	IO6 : NOP   0;
	      NOP   0;
	// --- FCM 07 - Recycling air flap ---
	    L "MAL1S032Par".Ilo.ILOMode;
	    L  7;
	    <>I;
	    SPB IO7;
	// man on
	      U     "MAL1S032Par".Ilo.GrCMDManOn[1];
	      S     "G273M".Gr.InManual; // RECYCLING AIR LOUVER KILN 1
	      S     "G278M".Gr.InManual; // WITHERING AIR KILN 1
	      R     "MAL1S032Par".Ilo.GrCMDManOn[1];
	// man off
	      U     "MAL1S032Par".Ilo.GrCMDManOff[1];
	      S     "G273M".Gr.CmdManualOff; // RECYCLING AIR LOUVER KILN 1
	      R     "G273M".Gr.InManual; // RECYCLING AIR LOUVER KILN 1
	      R     "G273M".USW14; // ILO-cmd
	      R     "G273M".USW15; // ILO-cmd
	      S     "G278M".Gr.CmdManualOff; // WITHERING AIR KILN 1
	      R     "G278M".Gr.InManual; // WITHERING AIR KILN 1
	      R     "G278M".USW14; // ILO-cmd
	      R     "G278M".USW15; // ILO-cmd
	      R     "MAL1S032Par".Ilo.GrCMDManOff[1];
	      R     "MAL1S032Par".Ilo.GrCMDManAdditional.Cmd1[1];
	      R     "MAL1S032Par".Ilo.GrCMDManAdditional.Cmd2[1];
	// man start
	      U     "MAL1S032Par".Ilo.GrCMDManStart[1];
	      S     "G273M".Gr.CmdOn; // RECYCLING AIR LOUVER KILN 1
	      S     "G273M".Gr.CmdContinue; // RECYCLING AIR LOUVER KILN 1
	      S     "G278M".Gr.CmdOn; // WITHERING AIR KILN 1
	      S     "G278M".Gr.CmdContinue; // WITHERING AIR KILN 1
	      R     "MAL1S032Par".Ilo.GrCMDManStart[1];
	      U     "MAL1S032Par".Ilo.GrCMDManStart[2];
	      R     "MAL1S032Par".Ilo.GrCMDManStart[2];
	// man stop
	      U     "MAL1S032Par".Ilo.GrCMDManStop[1];
	      S     "G273M".Gr.CmdOff; // RECYCLING AIR LOUVER KILN 1
	      S     "G278M".Gr.CmdOff; // WITHERING AIR KILN 1
	      R     "MAL1S032Par".Ilo.GrCMDManStop[1];
	// man fault reset
	      U     "MAL1S032Par".Ilo.GrCMDManFaultReset[1];
	      S     "G273M".Gr.CmdFaultReset; // RECYCLING AIR LOUVER KILN 1
	      S     "G278M".Gr.CmdFaultReset; // WITHERING AIR KILN 1
	      R     "MAL1S032Par".Ilo.GrCMDManFaultReset[1];
	// moving direction
	//
	// target position
	      UN    "G273M".Gr.InManual; // RECYCLING AIR LOUVER KILN 1
	      SPB   F07a;
	      L     "MAL1S032Par".Ilo.SetpointInt01[1];
	      T     "MAL1S032Par".Par.ParIntProcess.TarPos_ILO_RecycAir;
	F07a:  NOP   0;
	IO7 : NOP   0;
	      NOP   0;
	// --- FCM 09 - Floor drives ---
	    L "MAL1S032Par".Ilo.ILOMode;
	    L  9;
	    <>I;
	    SPB IO9;
	// man on
	      U     "MAL1S032Par".Ilo.GrCMDManOn[1];
	      S     "G266M".Gr.InManual; // TRAVELLING DRIVE KILN 1
	      R     "MAL1S032Par".Ilo.GrCMDManOn[1];
	// man off
	      U     "MAL1S032Par".Ilo.GrCMDManOff[1];
	      S     "G266M".Gr.CmdManualOff; // TRAVELLING DRIVE KILN 1
	      R     "G266M".Gr.InManual; // TRAVELLING DRIVE KILN 1
	      R     "G266M".USW14; // ILO-cmd
	      R     "G266M".USW15; // ILO-cmd
	      R     "MAL1S032Par".Ilo.GrCMDManOff[1];
	      R     "MAL1S032Par".Ilo.GrCMDManAdditional.Cmd1[1];
	      R     "MAL1S032Par".Ilo.GrCMDManAdditional.Cmd2[1];
	// man start
	      U     "MAL1S032Par".Ilo.GrCMDManStart[1];
	      S     "G266M".Gr.CmdOn; // TRAVELLING DRIVE KILN 1
	      S     "G266M".Gr.CmdContinue; // TRAVELLING DRIVE KILN 1
	      R     "MAL1S032Par".Ilo.GrCMDManStart[1];
	      U     "MAL1S032Par".Ilo.GrCMDManStart[2];
	      R     "MAL1S032Par".Ilo.GrCMDManStart[2];
	// man stop
	      U     "MAL1S032Par".Ilo.GrCMDManStop[1];
	      S     "G266M".Gr.CmdOff; // TRAVELLING DRIVE KILN 1
	      R     "MAL1S032Par".Ilo.GrCMDManStop[1];
	// man fault reset
	      U     "MAL1S032Par".Ilo.GrCMDManFaultReset[1];
	      S     "G266M".Gr.CmdFaultReset; // TRAVELLING DRIVE KILN 1
	      R     "MAL1S032Par".Ilo.GrCMDManFaultReset[1];
	f091: NOP   0;
	      UN    "G266M".Gr.InManual; // TRAVELLING DRIVE KILN 1
	      O     ;
	      UN    "MAL1S032Par".Ilo.GrCMDManAdditional.Cmd1[1];
	      UN    "MAL1S032Par".Ilo.GrCMDManAdditional.Cmd2[1];
	      SPB   f092;
	      U     "MAL1S032Par".Ilo.GrCMDManAdditional.Cmd1[1];
	      =     "G266M".USW14; // ILO-cmd run fwd
	      U     "MAL1S032Par".Ilo.GrCMDManAdditional.Cmd2[1];
	      =     "G266M".USW15; // ILO-cmd run rev
	// target position
	      L     "MAL1S032Par".Ilo.SetpointInt01[1];
	      T     "MAL1S032Par".Par.ParIntProcess.Speed_ILO_FloorRotating;
	f092: NOP   0;

	IO9 : NOP   0;
	      NOP   0;
	// --- FCM 10 - Floor drives and lifting devices ---
	    L "MAL1S032Par".Ilo.ILOMode;
	    L  10;
	    <>I;
	    SPB IO10;
	// man on
	      U     "MAL1S032Par".Ilo.GrCMDManOn[1];
	      S     "G265M".Gr.InManual; // LIFTING DEVICE KILN 1
	      S     "G265M".Gr.CmdOn; // No Button: LIFTING DEVICE KILN 1
	      S     "G265M".Gr.CmdContinue; // No Button LIFTING DEVICE KILN 1
	      S     "G266M".Gr.InManual; // TRAVELLING DRIVE KILN 1
	      R     "MAL1S032Par".Ilo.GrCMDManOn[1];
	// man off
	      U     "MAL1S032Par".Ilo.GrCMDManOff[1];
	      S     "G265M".Gr.CmdManualOff; // LIFTING DEVICE KILN 1
	      R     "G265M".Gr.InManual; // LIFTING DEVICE KILN 1
	      R     "G265M".USW14; // ILO-cmd
	      R     "G265M".USW15; // ILO-cmd
	      S     "G266M".Gr.CmdManualOff; // TRAVELLING DRIVE KILN 1
	      R     "G266M".Gr.InManual; // TRAVELLING DRIVE KILN 1
	      R     "G266M".USW14; // ILO-cmd
	      R     "G266M".USW15; // ILO-cmd
	      R     "MAL1S032Par".Ilo.GrCMDManOff[1];
	      R     "MAL1S032Par".Ilo.GrCMDManAdditional.Cmd1[1];
	      R     "MAL1S032Par".Ilo.GrCMDManAdditional.Cmd2[1];
	// man start
	      U     "MAL1S032Par".Ilo.GrCMDManStart[1];
	      S     "G266M".Gr.CmdOn; // TRAVELLING DRIVE KILN 1
	      S     "G266M".Gr.CmdContinue; // TRAVELLING DRIVE KILN 1
	      R     "MAL1S032Par".Ilo.GrCMDManStart[1];
	      U     "MAL1S032Par".Ilo.GrCMDManStart[2];
	      S     "G265M".Gr.CmdOn; // LIFTING DEVICE KILN 1
	      S     "G265M".Gr.CmdContinue; // LIFTING DEVICE KILN 1
	      R     "MAL1S032Par".Ilo.GrCMDManStart[2];
	      U     "MAL1S032Par".Ilo.GrCMDManStart[3];
	      R     "MAL1S032Par".Ilo.GrCMDManStart[3];
	// man stop
	      U     "MAL1S032Par".Ilo.GrCMDManStop[1];
	      S     "G265M".Gr.CmdOff; // LIFTING DEVICE KILN 1
	      S     "G266M".Gr.CmdOff; // TRAVELLING DRIVE KILN 1
	      R     "MAL1S032Par".Ilo.GrCMDManStop[1];
	// man fault reset
	      U     "MAL1S032Par".Ilo.GrCMDManFaultReset[1];
	      S     "G265M".Gr.CmdFaultReset; // LIFTING DEVICE KILN 1
	      S     "G266M".Gr.CmdFaultReset; // TRAVELLING DRIVE KILN 1
	      R     "MAL1S032Par".Ilo.GrCMDManFaultReset[1];
	// moving direction
	f101: NOP   0;
	      UN    "G266M".Gr.InManual; // TRAVELLING DRIVE KILN 1
	      O     ;
	      UN    "MAL1S032Par".Ilo.GrCMDManAdditional.Cmd1[1];
	      UN    "MAL1S032Par".Ilo.GrCMDManAdditional.Cmd2[1];
	      SPB   f102;
	      U     "MAL1S032Par".Ilo.GrCMDManAdditional.Cmd1[1];
	      =     "G266M".USW14; // ILO-cmd run fwd
	      U     "MAL1S032Par".Ilo.GrCMDManAdditional.Cmd2[1];
	      =     "G266M".USW15; // ILO-cmd run rev
	// target speed floor drives
	      L     "MAL1S032Par".Ilo.SetpointInt01[1];
	      T     "MAL1S032Par".Par.ParIntProcess.Speed_ILO_FloorRotating;
	f102: NOP   0;
	      UN    "G265M".Gr.InManual; // LIFTING DEVICE KILN 1
	      O(    ;
	      L     "MAL1S032Par".Ilo.Code_ILO_Funktion0;
	      L     1000;
	      <>I   ;
	      )     ;
	      SPB   f103;
	// target position lifting devices
	      L     "MAL1S032Par".Ilo.SetpointInt02[1];
	      T     "MAL1S032Par".Par.ParIntProcess.TarPos_ILO_LiftDev;
	f103: NOP   0;

	IO10 : NOP   0;
	      NOP   0;
	// --- FCM 11 - Floor drives and lifting devices and screw ---
	    L "MAL1S032Par".Ilo.ILOMode;
	    L  11;
	    <>I;
	    SPB IO11;
	// man on
	      U     "MAL1S032Par".Ilo.GrCMDManOn[1];
	      S     "G265M".Gr.InManual; // LIFTING DEVICE KILN 1
	      S     "G265M".Gr.CmdOn; // No Button: LIFTING DEVICE KILN 1
	      S     "G265M".Gr.CmdContinue; // No Button LIFTING DEVICE KILN 1
	      S     "G266M".Gr.InManual; // TRAVELLING DRIVE KILN 1
	      S     "G267M".Gr.InManual; // UNLOADING / LOADING SCREW KILN 1
	      R     "MAL1S032Par".Ilo.GrCMDManOn[1];
	// man off
	      U     "MAL1S032Par".Ilo.GrCMDManOff[1];
	      S     "G265M".Gr.CmdManualOff; // LIFTING DEVICE KILN 1
	      R     "G265M".Gr.InManual; // LIFTING DEVICE KILN 1
	      R     "G265M".USW14; // ILO-cmd
	      R     "G265M".USW15; // ILO-cmd
	      S     "G266M".Gr.CmdManualOff; // TRAVELLING DRIVE KILN 1
	      R     "G266M".Gr.InManual; // TRAVELLING DRIVE KILN 1
	      R     "G266M".USW14; // ILO-cmd
	      R     "G266M".USW15; // ILO-cmd
	      S     "G267M".Gr.CmdManualOff; // UNLOADING / LOADING SCREW KILN 1
	      R     "G267M".Gr.InManual; // UNLOADING / LOADING SCREW KILN 1
	      R     "G267M".USW14; // ILO-cmd
	      R     "G267M".USW15; // ILO-cmd
	      R     "MAL1S032Par".Ilo.GrCMDManOff[1];
	      R     "MAL1S032Par".Ilo.GrCMDManAdditional.Cmd1[1];
	      R     "MAL1S032Par".Ilo.GrCMDManAdditional.Cmd2[1];
	// man start
	      U     "MAL1S032Par".Ilo.GrCMDManStart[1];
	      S     "G266M".Gr.CmdOn; // TRAVELLING DRIVE KILN 1
	      S     "G266M".Gr.CmdContinue; // TRAVELLING DRIVE KILN 1
	      R     "MAL1S032Par".Ilo.GrCMDManStart[1];
	      U     "MAL1S032Par".Ilo.GrCMDManStart[2];
	      S     "G265M".Gr.CmdOn; // LIFTING DEVICE KILN 1
	      S     "G265M".Gr.CmdContinue; // LIFTING DEVICE KILN 1
	      R     "MAL1S032Par".Ilo.GrCMDManStart[2];
	      U     "MAL1S032Par".Ilo.GrCMDManStart[3];
	      S     "G267M".Gr.CmdOn; // UNLOADING / LOADING SCREW KILN 1
	      S     "G267M".Gr.CmdContinue; // UNLOADING / LOADING SCREW KILN 1
	      R     "MAL1S032Par".Ilo.GrCMDManStart[3];
	      U     "MAL1S032Par".Ilo.GrCMDManStart[4];
	      S     "G267M".Gr.CmdOn; // UNLOADING / LOADING SCREW KILN 1
	      S     "G267M".Gr.CmdContinue; // UNLOADING / LOADING SCREW KILN 1
	      R     "MAL1S032Par".Ilo.GrCMDManStart[4];
	// man stop
	      U     "MAL1S032Par".Ilo.GrCMDManStop[1];
	      S     "G265M".Gr.CmdOff; // LIFTING DEVICE KILN 1
	      S     "G266M".Gr.CmdOff; // TRAVELLING DRIVE KILN 1
	      S     "G267M".Gr.CmdOff; // UNLOADING / LOADING SCREW KILN 1
	      R     "MAL1S032Par".Ilo.GrCMDManStop[1];
	// man fault reset
	      U     "MAL1S032Par".Ilo.GrCMDManFaultReset[1];
	      S     "G265M".Gr.CmdFaultReset; // LIFTING DEVICE KILN 1
	      S     "G266M".Gr.CmdFaultReset; // TRAVELLING DRIVE KILN 1
	      S     "G267M".Gr.CmdFaultReset; // UNLOADING / LOADING SCREW KILN 1
	      R     "MAL1S032Par".Ilo.GrCMDManFaultReset[1];
	// moving direction
	      UN    "G266M".Gr.InManual; // TRAVELLING DRIVE KILN 1
	      O     ;
	      UN    "MAL1S032Par".Ilo.GrCMDManAdditional.Cmd1[1];
	      UN    "MAL1S032Par".Ilo.GrCMDManAdditional.Cmd2[1];
	      SPB   f112;
	      U     "MAL1S032Par".Ilo.GrCMDManAdditional.Cmd1[1];
	      =     "G266M".USW14; // ILO-cmd run fwd
	      U     "MAL1S032Par".Ilo.GrCMDManAdditional.Cmd2[1];
	      =     "G266M".USW15; // ILO-cmd run rev
	// target speed floor drives
	      L     "MAL1S032Par".Ilo.SetpointInt01[1];
	      T     "MAL1S032Par".Par.ParIntProcess.Speed_ILO_FloorRotating;
	f112: NOP   0;
	      UN    "G265M".Gr.InManual; // Malting Plant OAO Belsolod Ivanonvo Weissrussland
	      O(    ;
	      L     "MAL1S032Par".Ilo.Code_ILO_Funktion0;
	      L     1100;
	      <>I   ;
	      )     ;
	      SPB   f113;
	// target position lifting devices
	      L     "MAL1S032Par".Ilo.SetpointInt01[2];
	      L     "MAL1S032Par".Ilo.SetpointInt02[1];
	      T     "MAL1S032Par".Par.ParIntProcess.TarPos_ILO_LiftDev;
	f113: NOP   0;
	      UN    "G267M".Gr.InManual; // UNLOADING / LOADING SCREW KILN 1
	      O     ;
	      UN    "MAL1S032Par".Ilo.GrCMDManAdditional.Cmd1[3];
	      UN    "MAL1S032Par".Ilo.GrCMDManAdditional.Cmd2[3];
	      SPB   f114;
	      U     "MAL1S032Par".Ilo.GrCMDManAdditional.Cmd1[3];
	      =     "G267M".USW14; // ILO-cmd run fwd
	      U     "MAL1S032Par".Ilo.GrCMDManAdditional.Cmd2[3];
	      =     "G267M".USW15; // ILO-cmd run rev
	f114: NOP   0;
	IO11 : NOP   0;
	      NOP   0;
	// --- FCM 12 - Floor drives and lifting devices and screw and discharging flap ---
	    L "MAL1S032Par".Ilo.ILOMode;
	    L  12;
	    <>I;
	    SPB IO12;
	// man on
	      U     "MAL1S032Par".Ilo.GrCMDManOn[1];
	      S     "G265M".Gr.InManual; // LIFTING DEVICE KILN 1
	      S     "G265M".Gr.CmdOn; // No Button: LIFTING DEVICE KILN 1
	      S     "G265M".Gr.CmdContinue; // No Button LIFTING DEVICE KILN 1
	      S     "G266M".Gr.InManual; // TRAVELLING DRIVE KILN 1
	      S     "G267M".Gr.InManual; // UNLOADING / LOADING SCREW KILN 1
	      S     "G268M".Gr.InManual; // DISCHARGE DOOR KILN 1
	      R     "MAL1S032Par".Ilo.GrCMDManOn[1];
	// man off
	      U     "MAL1S032Par".Ilo.GrCMDManOff[1];
	      S     "G265M".Gr.CmdManualOff; // LIFTING DEVICE KILN 1
	      R     "G265M".Gr.InManual; // LIFTING DEVICE KILN 1
	      R     "G265M".USW14; // ILO-cmd
	      R     "G265M".USW15; // ILO-cmd
	      S     "G266M".Gr.CmdManualOff; // TRAVELLING DRIVE KILN 1
	      R     "G266M".Gr.InManual; // TRAVELLING DRIVE KILN 1
	      R     "G266M".USW14; // ILO-cmd
	      R     "G266M".USW15; // ILO-cmd
	      S     "G267M".Gr.CmdManualOff; // UNLOADING / LOADING SCREW KILN 1
	      R     "G267M".Gr.InManual; // UNLOADING / LOADING SCREW KILN 1
	      R     "G267M".USW14; // ILO-cmd
	      R     "G267M".USW15; // ILO-cmd
	      S     "G268M".Gr.CmdManualOff; // DISCHARGE DOOR KILN 1
	      R     "G268M".Gr.InManual; // DISCHARGE DOOR KILN 1
	      R     "G268M".USW14; // ILO-cmd
	      R     "G268M".USW15; // ILO-cmd
	      R     "MAL1S032Par".Ilo.GrCMDManOff[1];
	      R     "MAL1S032Par".Ilo.GrCMDManAdditional.Cmd1[1];
	      R     "MAL1S032Par".Ilo.GrCMDManAdditional.Cmd2[1];
	// man start
	      U     "MAL1S032Par".Ilo.GrCMDManStart[1];
	      S     "G266M".Gr.CmdOn; // TRAVELLING DRIVE KILN 1
	      S     "G266M".Gr.CmdContinue; // TRAVELLING DRIVE KILN 1
	      R     "MAL1S032Par".Ilo.GrCMDManStart[1];
	      U     "MAL1S032Par".Ilo.GrCMDManStart[2];
	      S     "G265M".Gr.CmdOn; // LIFTING DEVICE KILN 1
	      S     "G265M".Gr.CmdContinue; // LIFTING DEVICE KILN 1
	      R     "MAL1S032Par".Ilo.GrCMDManStart[2];
	      U     "MAL1S032Par".Ilo.GrCMDManStart[3];
	      S     "G267M".Gr.CmdOn; // UNLOADING / LOADING SCREW KILN 1
	      S     "G267M".Gr.CmdContinue; // UNLOADING / LOADING SCREW KILN 1
	      R     "MAL1S032Par".Ilo.GrCMDManStart[3];
	      U     "MAL1S032Par".Ilo.GrCMDManStart[4];
	      S     "G267M".Gr.CmdOn; // UNLOADING / LOADING SCREW KILN 1
	      S     "G267M".Gr.CmdContinue; // UNLOADING / LOADING SCREW KILN 1
	      R     "MAL1S032Par".Ilo.GrCMDManStart[4];
	// man stop
	      U     "MAL1S032Par".Ilo.GrCMDManStop[1];
	      S     "G265M".Gr.CmdOff; // LIFTING DEVICE KILN 1
	      S     "G266M".Gr.CmdOff; // TRAVELLING DRIVE KILN 1
	      S     "G267M".Gr.CmdOff; // UNLOADING / LOADING SCREW KILN 1
	      S     "G268M".Gr.CmdOff; // DISCHARGE DOOR KILN 1
	      R     "MAL1S032Par".Ilo.GrCMDManStop[1];
	// man fault reset
	      U     "MAL1S032Par".Ilo.GrCMDManFaultReset[1];
	      S     "G265M".Gr.CmdFaultReset; // LIFTING DEVICE KILN 1
	      S     "G266M".Gr.CmdFaultReset; // TRAVELLING DRIVE KILN 1
	      S     "G267M".Gr.CmdFaultReset; // UNLOADING / LOADING SCREW KILN 1
	      S     "G268M".Gr.CmdFaultReset; // DISCHARGE DOOR KILN 1
	      R     "MAL1S032Par".Ilo.GrCMDManFaultReset[1];
	// moving direction
	      UN    "G266M".Gr.InManual; // TRAVELLING DRIVE KILN 1
	      O     ;
	      UN    "MAL1S032Par".Ilo.GrCMDManAdditional.Cmd1[1];
	      UN    "MAL1S032Par".Ilo.GrCMDManAdditional.Cmd2[1];
	      SPB   f122;
	      U     "MAL1S032Par".Ilo.GrCMDManAdditional.Cmd1[1];
	      =     "G266M".USW14; // ILO-cmd run fwd
	      U     "MAL1S032Par".Ilo.GrCMDManAdditional.Cmd2[1];
	      =     "G266M".USW15; // ILO-cmd run rev
	// target speed floor drives
	      L     "MAL1S032Par".Ilo.SetpointInt01[1];
	      T     "MAL1S032Par".Par.ParIntProcess.Speed_ILO_FloorRotating;
	f122: NOP   0;
	      UN    "G265M".Gr.InManual; // LIFTING DEVICE KILN 1
	      O(    ;
	      L     "MAL1S032Par".Ilo.Code_ILO_Funktion0;
	      L     1200;
	      <>I   ;
	      )     ;
	      SPB   f123;
	// target position lifting devices
	      L     "MAL1S032Par".Ilo.SetpointInt02[1];
	      T     "MAL1S032Par".Par.ParIntProcess.TarPos_ILO_LiftDev;
	f123: NOP   0;
	      UN    "G267M".Gr.InManual; // Malting Plant OAO Belsolod Ivanonvo Weissrussland
	      O     ;
	      UN    "MAL1S032Par".Ilo.GrCMDManAdditional.Cmd1[3];
	      UN    "MAL1S032Par".Ilo.GrCMDManAdditional.Cmd2[3];
	      SPB   f124;
	      U     "MAL1S032Par".Ilo.GrCMDManAdditional.Cmd1[3];
	      =     "G267M".USW14; // ILO-cmd run fwd
	      U     "MAL1S032Par".Ilo.GrCMDManAdditional.Cmd2[3];
	      =     "G267M".USW15; // ILO-cmd run rev
	f124: NOP   0;
	      UN    "G268M".Gr.InManual; // DISCHARGE DOOR KILN 1
	      O     ;
	      UN    "MAL1S032Par".Ilo.GrCMDManAdditional.Cmd1[4];
	      UN    "MAL1S032Par".Ilo.GrCMDManAdditional.Cmd2[4];
	      SPB   f125;
	      U     "MAL1S032Par".Ilo.GrCMDManAdditional.Cmd1[4];
	      =     "G268M".USW14; // ILO-cmd OPEN
	      U     "MAL1S032Par".Ilo.GrCMDManAdditional.Cmd2[4];
	      =     "G268M".USW15; // ILO-cmd CLOSE
	f125: NOP   0;
	IO12 : NOP   0;
	//
	// copy state
	      U     "G265M".Gr.InOutAutostartMan; // LIFTING DEVICE KILN 1
	      =     "MAL1S032Par".Ilo.GrSTMan[1];
	      U     "G266M".Gr.InOutAutostartMan; // TRAVELLING DRIVE KILN 1
	      =     "MAL1S032Par".Ilo.GrSTMan[2];
	      U     "G267M".Gr.InOutAutostartMan; // UNLOADING / LOADING SCREW KILN 1
	      =     "MAL1S032Par".Ilo.GrSTMan[3];
	      U     "G268M".Gr.InOutAutostartMan; // DISCHARGE DOOR KILN 1
	      =     "MAL1S032Par".Ilo.GrSTMan[4];
	      U     "G271M".Gr.InOutAutostartMan; // FAN KILN 1
	      =     "MAL1S032Par".Ilo.GrSTMan[6];
	      U     "G276M".Gr.InOutAutostartMan; // HEATING KILN 1
	      =     "MAL1S032Par".Ilo.GrSTMan[11];
	      U     "G277M".Gr.InOutAutostartMan; // LOUVER AIR HEATER 1 FOR KILN 1
	      =     "MAL1S032Par".Ilo.GrSTMan[12];
	      U     "G272M".Gr.InOutAutostartMan; // FRESH AIR LOUVER KILN 1
	      =     "MAL1S032Par".Ilo.GrSTMan[13];
	      U     "G278M".Gr.InOutAutostartMan; // WITHERING AIR KILN 1
	      =     "MAL1S032Par".Ilo.GrSTMan[14];
	      U     "G273M".Gr.InOutAutostartMan; // RECYCLING AIR LOUVER KILN 1
	      =     "MAL1S032Par".Ilo.GrSTMan[15];
	      U     "G279M".Gr.InOutAutostartMan; // HEATING KILN 1 + 2
	      =     "MAL1S032Par".Ilo.GrSTMan[16];
	NETWORK
	TITLE =ASW_9999: Init Flag
	// clear all flags explicde to find them back
	      U     "MAL1S032".PCRead.Step.StIdling;
	      O     "MAL1S032".PCRead.Step.StPassive;
	      R     "MAL1S032Par".Par.FlagFunction_1.StepLoading;
	      R     "MAL1S032Par".Par.FlagFunction_1.StepUnloading;
	      R     "MAL1S032Par".Par.FlagFunction_1.StepCleaning;
	      R     "MAL1S032Par".Par.FlagFunction_1.LoadingBreak;
	      R     "MAL1S032Par".Par.FlagFunction_1.UnloadingBreak;
	      R     "MAL1S032Par".Par.FlagFunction_1.CleaningBreak;
	      R     "MAL1S032Par".Par.FlagFunction_1.FinishLoading;
	      R     "MAL1S032Par".Par.FlagFunction_1.FinishUnloading;
	      R     "MAL1S032Par".Par.FlagFunction_1.FinishCleaning;
	      R     "MAL1S032Par".Par.FlagFunction_1.Entladerunden_erreicht;
	      R     "MAL1S032Par".Par.FlagFunction_1.Reinigungsrunde_erreicht;
	      R     "MAL1S032Par".Par.FlagFunction_1.UnloadEnd;
	      R     "MAL1S032Par".Par.FlagFunction_1.LoadEnd;
	      R     "MAL1S032Par".Par.FlagFunction_1.UnloadFirstPart;
	      R     "MAL1S032Par".Par.FlagFunction_1.UnloadSecondPart;
	      R     "MAL1S032Par".Par.FlagProcess.ProcessActive;
	      R     "MAL1S032Par".Par.FlagProcess.StartProzess_FP;
	      R     "MAL1S032Par".Par.FlagProcess.StartProzess_SCAN;
	      R     "MAL1S032Par".Par.FlagProcess.TurningFloor;
	      R     "MAL1S032Par".Par.FlagProcess.Cooling_Activ;
	      R     "MAL1S032Par".Par.FlagProcess.FP_SendResultToPIC;
	      R     "MAL1S032Par".Par.FlagProcess.ProcessEnd;

	NETWORK
	TITLE =Main0_End: Init flag
		SET;
		R     MAL1S032.Gr.All.CmdNewSelection;
		R     MAL1S032.ToASW.CmdNewBatch;
		R     MAL1S032.ToASW.CmdModify;

	NETWORK
	TITLE =End of block

	      BE    ;

	END_FUNCTION
